// TIA Portal V19 export
DATA_BLOCK "An Scale2"   // DB6
// stored: InstanceOfName An Scaling, InstanceOfType FB
"An Scaling"
   // VAR_INPUT
   //    "Sensor IN" : Int;
   //    "Analog Min" { ExternalAccessible := 'False'; ExternalVisible := 'False'; ExternalWritable := 'False'} : Int;
   //    "Analog Max" { ExternalAccessible := 'False'; ExternalVisible := 'False'; ExternalWritable := 'False'} : Int;
   //    "Scaled Min" { ExternalAccessible := 'False'; ExternalVisible := 'False'; ExternalWritable := 'False'} : Real;
   //    "Scaled Max" { ExternalAccessible := 'False'; ExternalVisible := 'False'; ExternalWritable := 'False'} : Real;
   // END_VAR
   // VAR_OUTPUT
   //    Scaled_Sensor : Real;
   // END_VAR
   // VAR
   //    Normalised_sensor { ExternalAccessible := 'False'; ExternalVisible := 'False'; ExternalWritable := 'False'} : Real;
   //    sensor_result { ExternalAccessible := 'False'; ExternalVisible := 'False'; ExternalWritable := 'False'} : Int;
   // END_VAR
BEGIN
END_DATA_BLOCK
